// TIA Portal project "Ares_URC_PLC" (V11)

(* hardware
DEVICE "SIMATIC 1200 station_1"  S71200.Device
   slot 0: "S7-1200 rack"  Rack  V1.0
   slot 1: "PLC_1"  CPU 1215C DC/DC/DC  6ES7 215-1AG31-0XB0  V3.0
   slot 101: "CM 1241 (RS422/485)_1"  6ES7 241-1CH31-0XB0  V1.0
*)

// ===== PLC "PLC_1"  CPU 1215C DC/DC/DC =====

VAR_GLOBAL   // PLC tag table "Default tag table"
   "Tag_1" AT %M1.0 : Bool;
   "System_Byte" AT %MB1 : Byte;
   "DiagStatusUpdate" AT %M1.1 : Bool;
   "AlwaysTRUE" AT %M1.2 : Bool;
   "AlwaysFALSE" AT %M1.3 : Bool;
END_VAR

DATA_BLOCK "ModbusRTU"   // DB1
{ S7_Optimized_Access := 'FALSE' }
VERSION : 0.1
   VAR
      RequestSettings : Bool;
      SettingsDone : Bool;
      SettingsError : Bool;
      "SettingsErrorStatus]" : Word;
      RequestTransfer : Bool;
      RequestSlaveAdress : UInt;
      RequestTransferMode : USInt;
      RequestDataAddress : UDInt;
      RequestDataLength : UInt;
      RequestDone : Bool;
      RequestBusy : Bool;
      RequestError : Bool;
      RequestErrorStatus : Word;
      RequestActualRegisterBank : VREF;
      RequestRegistersRTU_ML1 : Array [1 .. 100] of Word;
      RequestRegistersRTU_ML2 : Array [1 .. 100] of Word;
      RequestRegistersRTU_ML3 : Array [1 .. 100] of Word;
      RequestRegistersRTU_MR1 : Array [1 .. 100] of Word;
      RequestRegistersRTU_MR2 : Array [1 .. 100] of Word;
      RequestRegistersRTU_MR3 : Array [1 .. 100] of Word;
   END_VAR
BEGIN
END_DATA_BLOCK

DATA_BLOCK "ModbusTCP"   // DB2
{ S7_Optimized_Access := 'FALSE' }
VERSION : 0.1
BEGIN
END_DATA_BLOCK

DATA_BLOCK "FBModbusRTU_DB"   // DB5
{ S7_Optimized_Access := 'FALSE' }
VERSION : 0.1
// stored: InstanceOfName FBModbusRTU
"FBModbusRTU"
BEGIN
END_DATA_BLOCK

FUNCTION_BLOCK "FBModbusRTU"   // FB1, LAD
{ S7_Optimized_Access := 'FALSE' }
VERSION : 0.1
BEGIN

REGION Network 1
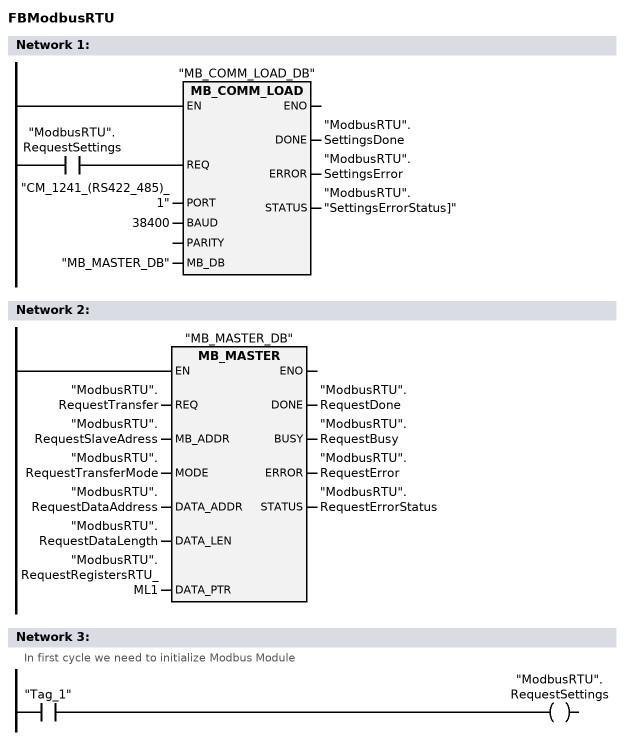
   "MB_COMM_LOAD_DB"(REQ := "ModbusRTU".RequestSettings,   // MB_COMM_LOAD
                     PORT := "CM_1241_(RS422_485)_1",
                     BAUD := 38400,
                     MB_DB := "MB_MASTER_DB",
                     DONE => "ModbusRTU".SettingsDone,
                     ERROR => "ModbusRTU".SettingsError,
                     STATUS => "ModbusRTU"."SettingsErrorStatus]");
END_REGION

REGION Network 2
   "MB_MASTER_DB"(REQ := "ModbusRTU".RequestTransfer,   // MB_MASTER
                  MB_ADDR := "ModbusRTU".RequestSlaveAdress,
                  MODE := "ModbusRTU".RequestTransferMode,
                  DATA_ADDR := "ModbusRTU".RequestDataAddress,
                  DATA_LEN := "ModbusRTU".RequestDataLength,
                  DATA_PTR := "ModbusRTU".RequestRegistersRTU_ML1,
                  DONE => "ModbusRTU".RequestDone,
                  BUSY => "ModbusRTU".RequestBusy,
                  ERROR => "ModbusRTU".RequestError,
                  STATUS => "ModbusRTU".RequestErrorStatus);
END_REGION

REGION Network 3
   // In first cycle we need to initialize Modbus Module
   RUNG wire#powerrail
      Contact( "Tag_1" )
      Coil( "ModbusRTU".RequestSettings )
   END_RUNG
   // the same network as SCL:
   "ModbusRTU".RequestSettings := "Tag_1";
END_REGION
END_FUNCTION_BLOCK

ORGANIZATION_BLOCK "Main"   // OB1, LAD, ProgramCycle
TITLE = "Main Program Sweep (Cycle)"
{ S7_Optimized_Access := 'FALSE' }
VERSION : 0.1
BEGIN

REGION Network 1
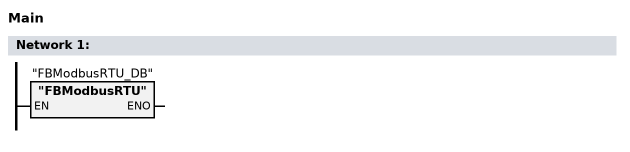
   RUNG wire#powerrail
      "FBModbusRTU_DB"()
   END_RUNG
   // the same network as SCL:
   "FBModbusRTU_DB"();   // "FBModbusRTU"
END_REGION
END_ORGANIZATION_BLOCK